SUBAPPLICATION Uebung_10c4_sub (* SoftKey_F1/_F2 auf DigitalOutput_Q1/_Q2 mit GreenWhiteBackground mit Typed Subapp *)
  (* Standard: 61499-2 *)
  (* Version 1.0, 2025-07-26, franz *)
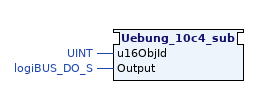
  VAR_INPUT
    u16ObjId : UINT := isobus::ID_NULL; (* Object ID *)
    Output : logiBUS_DO_S := logiBUS_DO::Invalid; (* Identify the Output Output_Q1..Q8 *)
  END_VAR
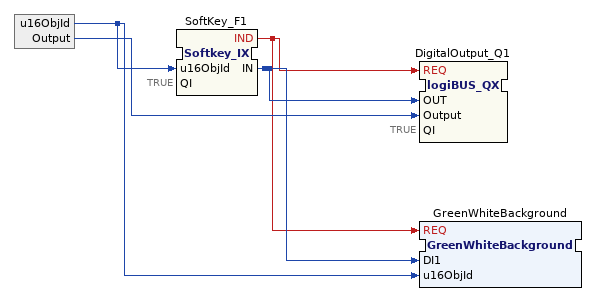
  FBS
    DigitalOutput_Q1 : logiBUS_QX(QI := TRUE);
    SoftKey_F1 : Softkey_IX(QI := TRUE);
  END_FBS
  SUBAPPS
    GreenWhiteBackground : GreenWhiteBackground;
  END_SUBAPPS
  EVENT_CONNECTIONS
    SoftKey_F1.IND TO GreenWhiteBackground.REQ;
    SoftKey_F1.IND TO DigitalOutput_Q1.REQ;
  END_CONNECTIONS
  DATA_CONNECTIONS
    SoftKey_F1.IN TO GreenWhiteBackground.DI1;
    SoftKey_F1.IN TO DigitalOutput_Q1.OUT;
    u16ObjId TO SoftKey_F1.u16ObjId;
    u16ObjId TO GreenWhiteBackground.u16ObjId;
    Output TO DigitalOutput_Q1.Output;
  END_CONNECTIONS
END_SUBAPPLICATION
